{attribute 'qualified_only'}
VAR_GLOBAL
	mb_Input_Coils : ARRAY [0..3] OF BOOL;
	mb_Output_Coils : ARRAY [0..7] OF BOOL;
END_VAR

(* stored: Version 1.1.0.1, ProductVersion 3.1.4024.12
   GVL GVL: Id {8494bc1c-1164-499e-8085-e7e68ec3da00} *)
